FUNCTION F_ConfigPositionEmulation_002

END_FUNCTION

(* stored: Version 1.1.0.1, ProductVersion 3.1.4024.9
   POU F_ConfigPositionEmulation_002: Id {68c4d31b-ce0b-4a5c-8e38-919ceb2ce310}, SpecialFunc None *)
